FUNCTION_BLOCK fb_vacuumRetry
VAR_INPUT
	in_flg_run: BOOL;
END_VAR
VAR_OUTPUT
	out_flg_faied: BOOL;
	out_flg_Done: BOOL;
END_VAR
VAR
	fbi_flg_run: R_TRIG;
	var_process: INT;
	var_retryTimes: INT;
	flg_chuckDone: BOOL;
	flg_pushDone: BOOL;
END_VAR

fbi_flg_run(CLK:= in_flg_run, Q=> );
IF fbi_flg_run.Q  THEN
	var_process := 1;
END_IF
IF NOT in_flg_run THEN
	out_flg_done := FALSE;
	out_flg_faied := FALSE;
	flg_chuckDone := FALSE;
	flg_pushDone := FALSE;
	var_retryTimes := 0;
END_IF
CASE var_process OF 
	1:
		gvl_axis.fbi_motionControler.in_flg_start := FALSE;
		gvl_axis.fbi_motionControler.in_var_targetPosX := gvl_param.var_productInfo[gvl_param.var_currentProductID].teachPos.pickUp.x;
		gvl_axis.fbi_motionControler.in_var_targetPosY := gvl_param.var_productInfo[gvl_param.var_currentProductID].teachPos.pickUp.y;
		gvl_axis.fbi_motionControler.in_var_targetPosZ := gvl_param.var_productInfo[gvl_param.var_currentProductID].teachPos.pickUp.z;
		gvl_axis.fbi_motionControler.in_var_direction := eP_motionDirection.XYZ;
		gvl_solv.fbi_chuck.in_flg_run := FALSE;
		gvl_solv.fbi_chuck.in_var_moveMode := eP_svMoveMode.svB;
		gvl_solv.fbi_push.in_flg_run := FALSE;
		gvl_solv.fbi_push.in_var_moveMode := eP_svMoveMode.svB;
		flg_chuckDone := FALSE;
		flg_pushDone := FALSE;
		var_process := 2;
	2:
		gvl_solv.fbi_push.in_flg_run := TRUE;
		gvl_solv.fbi_chuck.in_flg_run := TRUE;
		var_process := 3;
	3:
		IF gvl_solv.fbi_chuck.out_flg_Done THEN
			flg_chuckDone := TRUE;
		END_IF
		IF gvl_solv.fbi_push.out_flg_Done THEN
			flg_pushDone := TRUE;
		END_IF
		IF flg_pushDone AND flg_chuckDone THEN
			gvl_axis.fbi_motionControler.in_flg_start := TRUE;
			var_process := 4;
		END_IF
	4:
		IF gvl_axis.fbi_motionControler.out_flg_Done THEN
			gvl_axis.fbi_motionControler.in_flg_start := FALSE;
			var_process := 5;
		END_IF
	5:
		gvl_axis.fbi_motionControler.in_flg_start := FALSE;
		gvl_axis.fbi_motionControler.in_var_targetPosX := gvl_param.var_productInfo[gvl_param.var_currentProductID].teachPos.initial.x;
		gvl_axis.fbi_motionControler.in_var_targetPosY := gvl_param.var_productInfo[gvl_param.var_currentProductID].teachPos.initial.y;
		gvl_axis.fbi_motionControler.in_var_targetPosZ := gvl_param.var_productInfo[gvl_param.var_currentProductID].teachPos.initial.z;
		gvl_axis.fbi_motionControler.in_var_direction := eP_motionDirection.ZYX;
		gvl_solv.fbi_chuck.in_flg_run := FALSE;
		gvl_solv.fbi_chuck.in_var_moveMode := eP_svMoveMode.svA;
		gvl_solv.fbi_push.in_flg_run := FALSE;
		gvl_solv.fbi_push.in_var_moveMode := eP_svMoveMode.svA;
		flg_chuckDone := FALSE;
		flg_pushDone := FALSE;
		var_process := 6;
	6:
		gvl_solv.fbi_chuck.in_flg_run := TRUE;
		gvl_solv.fbi_push.in_flg_run := TRUE;
		IF gvl_solv.fbi_chuck.out_flg_Done THEN
			flg_chuckDone := TRUE;
		END_IF
		IF gvl_solv.fbi_push.out_flg_Done THEN
			flg_pushDone := TRUE;
		END_IF
		IF flg_pushDone AND flg_chuckDone THEN
			gvl_axis.fbi_motionControler.in_flg_start := TRUE;
			var_process := 7;
		END_IF
	7:
		IF gvl_axis.fbi_motionControler.out_flg_Done THEN
			gvl_axis.fbi_motionControler.in_flg_start := FALSE;
			var_process := 8;
		END_IF
	8:
		IF gvl_solv.ref_ejector.input.in_flg_sensVac THEN
			var_process := 20;
		ELSE
			var_process := 9;
		END_IF
	9:
		IF var_retryTimes < 3 THEN
			var_retryTimes := var_retryTimes + 1;
			var_process := 1;
		ELSE
			gvl_solv.fbi_ejector.in_flg_run := FALSE;
			gvl_solv.fbi_ejector.in_var_vacMode := eP_ejevacMode.vacON;
			var_process := 10;
		END_IF
	10:
		gvl_solv.fbi_ejector.in_flg_run := TRUE;
		var_process := 11;
	20:
	
		out_flg_Done := TRUE;
		var_process := 21;
	21:
		out_flg_Done := FALSE;
END_CASE

END_FUNCTION_BLOCK

(* stored: Version 1.1.0.1, ProductVersion 3.1.4024.11
   POU fb_vacuumRetry: Id {6c7fb780-0775-42c1-93d5-a5c9daeec520}, SpecialFunc None *)
